TYPE ST_AX8108 :
STRUCT
	
	//M1 Motor Structure
	iPosition								AT %I*		: LREAL;
	iStatusWord								AT %I*		: UINT;
	qControlWord							AT %Q*		: UINT;
	qTargetVelocity							AT %Q*		: LREAL;
	nState									AT %I*		: UINT;						//Terminal State from IO Terminal Info Data
	sStatus												: STRING(200);
	Axis                                        	 	: AXIS_REF; 				//Motor M1 Seal Stage Vertical Axis
	n_AxisTorqueLimitation					AT %Q*		: UINT		:=	32767;
	n_AxisActualTorque									: REAL; 					// now part of structured varaible axis_ref

	//M1 Motor Safety
	bTS_Run									AT %Q*		: BOOL;
	bTS_ErrorAck							AT %Q*		: BOOL;

END_STRUCT
END_TYPE

(* stored: Version 1.1.0.1, ProductVersion 3.1.4024.12
   DUT ST_AX8108: Id {27df3599-5884-4e9c-845c-1a13e5935d53} *)
